// TIA Portal V19 export
ORGANIZATION_BLOCK "A03_OB32_CyclicInterrupt"   // OB32, LAD, CyclicInterrupt
// stored: AutoNumber false, SetENOAutomatically false
   VAR_INPUT
      Initial_Call : Bool;   // Initial call of this OB
      Event_Count : Int;   // Events discarded
   END_VAR
BEGIN

REGION Network 1
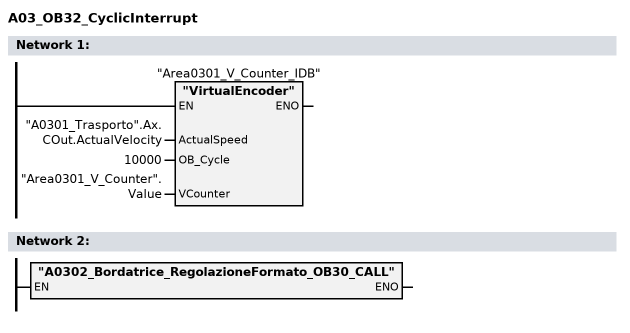
   RUNG wire#powerrail
      "Area0301_V_Counter_IDB"(ActualSpeed := "A0301_Trasporto".Ax.COut.ActualVelocity, OB_Cycle := 10000, VCounter := "Area0301_V_Counter".Value)
   END_RUNG
   // the same network as SCL:
   "Area0301_V_Counter_IDB"(ActualSpeed := "A0301_Trasporto".Ax.COut.ActualVelocity,   // "VirtualEncoder"
                           OB_Cycle := 10000,
                           VCounter := "Area0301_V_Counter".Value);
END_REGION

REGION Network 2
   RUNG wire#powerrail
      "A0302_Bordatrice_RegolazioneFormato_OB30_CALL"()
   END_RUNG
   // the same network as SCL:
   "A0302_Bordatrice_RegolazioneFormato_OB30_CALL"();
END_REGION
END_ORGANIZATION_BLOCK
